{attribute 'linkalways'} 
{attribute 'no_explicit_call' := 'This FB is a CLASS and must be accessed using methods or properties'}
{attribute 'enable_dynamic_creation'}
FUNCTION_BLOCK _FLOAT EXTENDS AliasDatatypeBase
VAR
	localData : FLOAT;
	activeData : REFERENCE TO FLOAT REF= localData;
	aliasBaseDatatype : _LREAL(localData);
END_VAR

PROPERTY PUBLIC Address : PVOID
GET
Address := ADR(activeData);
END_GET
END_PROPERTY

METHOD PUBLIC ClearReference
VAR_INPUT
END_VAR
activeData REF= localData;
SetBaseDatatypeReference();
END_METHOD

METHOD PUBLIC Clone : I_Datatype
VAR
    pClone : POINTER TO _FLOAT;
END_VAR
pClone := __NEW(_FLOAT(InitialValue := Value));
Clone := pClone^;
END_METHOD

METHOD FB_init : BOOL
VAR_INPUT
	bInitRetains : BOOL; // if TRUE, the retain variables are initialized (warm start / cold start)
	bInCopyCode : BOOL;  // if TRUE, the instance afterwards gets moved into the copy code (online change)
	InitialValue : FLOAT;
END_VAR
localData := InitialValue;
SetBaseDatatypeReference();
AddBaseDatatype(aliasBaseDatatype);
END_METHOD

PROPERTY PUBLIC Identifier : T_MAXSTRING
GET
Identifier := 'FLOAT';
END_GET
END_PROPERTY

METHOD PUBLIC MakeReferenceTo
VAR_INPUT
	ReferenceTarget : REFERENCE TO FLOAT;
END_VAR
activeData REF= ReferenceTarget;
SetBaseDatatypeReference();
END_METHOD

METHOD PROTECTED SetBaseDatatypeReference
VAR_INPUT
END_VAR
aliasBaseDatatype.MakeReferenceTo(activeData);
END_METHOD

PROPERTY PUBLIC Size : UDINT
GET
Size := SIZEOF(activeData);
END_GET
END_PROPERTY

METHOD TryMakeReferenceTo : BOOL
VAR_INPUT
	Target : I_Datatype;
END_VAR
VAR
	targetAsAlias : I_AliasDatatype;
	pTargetData : POINTER TO FLOAT;
END_VAR
IF NOT Target.TryResolveAsAliasDatatype(targetAsAlias) THEN
	RETURN;
END_IF

IF targetAsAlias.Identifier <> Identifier THEN
	RETURN;
END_IF

pTargetData := Target.Address;
activeData REF= pTargetData^;
SetBaseDatatypeReference();
TryMakeReferenceTo := TRUE;
END_METHOD

PROPERTY PUBLIC Value : FLOAT
GET
Value := activeData;
END_GET
SET
activeData := Value;
END_SET
END_PROPERTY

END_FUNCTION_BLOCK

(* stored: Version 1.1.0.1, ProductVersion 3.1.4024.12
   POU _FLOAT: Id {ff4acc88-b4ef-039e-2595-847ea4a548ba}, SpecialFunc None
   Folder Constructor: Id {412e582f-94b8-092c-3cb8-c4207291a193}
   Folder Protected: Id {81b92b6e-4201-0ee5-3799-a6ee2a4eec80}
   Property Address: Id {3d7d18b1-2d73-02dc-0ea6-15422d947978}
   Get Get: Id {06ca092b-79cb-0912-3812-8268eceb65e9}
   Method ClearReference: Id {beb9094b-dec0-0ad6-3309-0481956e1c22}
   Method Clone: Id {a8938d8d-a0e1-0001-24a3-c62368fc7a6b}
   Method FB_init: Id {964f2a87-c7a3-0e9b-3938-ccf0f38265c7}
   Property Identifier: Id {1632188e-cea2-0d94-1a05-611820c29699}
   Get Get: Id {f7f3dbfb-7e30-0c10-3aa9-e0ac0f6cc979}
   Method MakeReferenceTo: Id {edf21b22-15a6-0dc7-1c3f-6fe0e39a444f}
   Method SetBaseDatatypeReference: Id {5df21de2-bd74-0f5c-0a76-53dc1bcde600}
   Property Size: Id {9a36642e-b334-079d-099a-fb042f122e9c}
   Get Get: Id {e7a88d05-bd27-0421-3101-695d35bf781b}
   Method TryMakeReferenceTo: Id {66ad58ca-4cff-0fad-182f-2c82500eccd2}
   Property Value: Id {1fb88f68-b0c5-0296-0f56-a8d9ae759e6b}
   Get Get: Id {8bdcb384-8a67-022d-038b-52ee13c95a00}
   Set Set: Id {5795a749-afad-022f-1a63-33b91eec5eb2} *)
